{attribute 'qualified_only'}
VAR_GLOBAL CONSTANT
	 ROBOT_RADIUS : LREAL := 0.15;		  // in m
	 RING_SIZE : INT := 60;
END_VAR

(* stored: Version 1.1.0.1, ProductVersion 3.1.4026.13
   GVL GVL: Id {5a12a4ab-ceee-4884-9e65-7f3189ae7563} *)
